SUBAPPLICATION Uebung_004b (* Toggle Flip-Flop mit IE / Split *)
  (* Standard: 61499-2 *)
  (* Version 1.0, 2023-10-23, franz *)
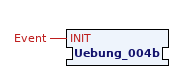
  EVENT_INPUT
    INIT;
  END_EVENT
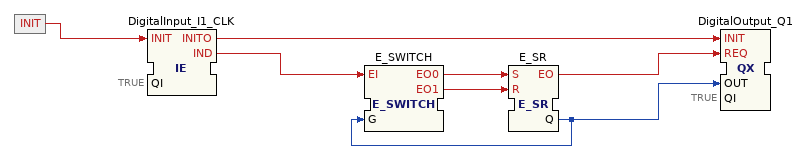
  FBS
    DigitalOutput_Q1 : QX(QI := TRUE);
    DigitalInput_I1_CLK : IE(QI := TRUE);
    E_SR : E_SR;
    E_SWITCH : E_SWITCH;
  END_FBS
  EVENT_CONNECTIONS
    INIT TO DigitalInput_I1_CLK.INIT;
    DigitalInput_I1_CLK.INITO TO DigitalOutput_Q1.INIT;
    E_SR.EO TO DigitalOutput_Q1.REQ;
    E_SWITCH.EO0 TO E_SR.S;
    E_SWITCH.EO1 TO E_SR.R;
    DigitalInput_I1_CLK.IND TO E_SWITCH.EI;
  END_CONNECTIONS
  DATA_CONNECTIONS
    E_SR.Q TO DigitalOutput_Q1.OUT;
    E_SR.Q TO E_SWITCH.G;
  END_CONNECTIONS
END_SUBAPPLICATION
